Yaskawa INFORM job: kufsatest1_01_01_23_10_57.JBI

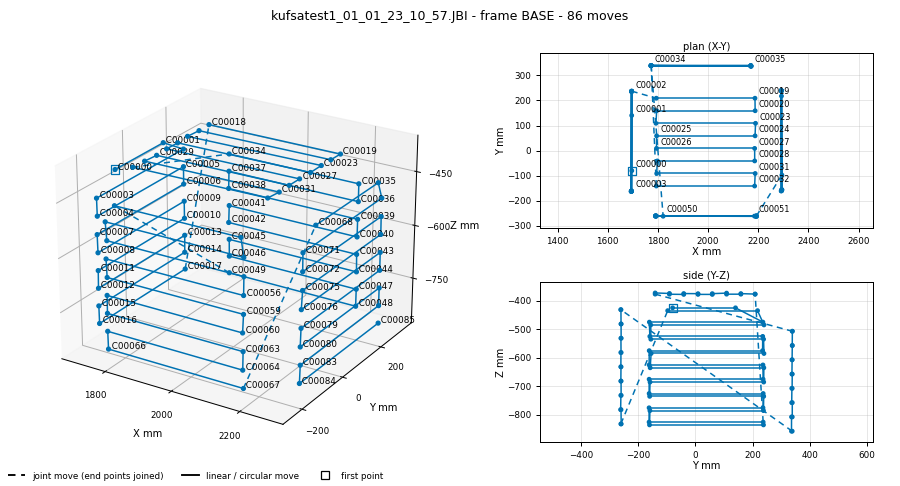
[picture p0: tool path of kufsatest1_01_01_23_10_57.JBI in frame BASE, 86 of 86 moves have a stored position in this frame; points joined in program order, loops and branches not executed]
/JOB
//NAME kufsa_test
//POS
///NPOS 86,0,0,0,0,0
///TOOL 0
///POSTYPE BASE
///RECTAN
///RCONF 1,0,0,0,0,0,0,0,0,0,0,0,0,0,0,0,0,0,0,0,0,0,0,0
C00000=1696.132000,-80.047400,-425.128800,0.000000,90.000000,0.000000
C00001=1695.649900,140.027500,-425.128800,0.000000,90.000000,0.000000
C00002=1695.009700,236.007500,-475.128800,0.000000,90.000000,0.000000
C00003=1694.894300,-161.509200,-475.128800,0.000000,90.000000,0.000000
C00004=1694.500400,-159.876400,-525.128800,0.000000,90.000000,0.000000
C00005=1694.957700,235.269700,-525.128800,0.000000,90.000000,0.000000
C00006=1695.172400,234.870300,-575.128800,0.000000,90.000000,0.000000
C00007=1694.072400,-162.036300,-575.128800,0.000000,90.000000,0.000000
C00008=1695.266200,-162.303200,-625.128800,0.000000,90.000000,0.000000
C00009=1695.465900,236.123700,-625.128800,0.000000,90.000000,0.000000
C00010=1695.422700,236.644700,-675.128800,0.000000,90.000000,0.000000
C00011=1694.457900,-162.352100,-675.128800,0.000000,90.000000,0.000000
C00012=1693.613400,-162.296700,-725.128800,0.000000,90.000000,0.000000
C00013=1695.359600,236.966000,-725.128800,0.000000,90.000000,0.000000
C00014=1695.305600,236.328100,-775.128800,0.000000,90.000000,0.000000
C00015=1693.299800,-162.503900,-775.128800,0.000000,90.000000,0.000000
C00016=1694.079700,-162.510900,-825.128800,0.000000,90.000000,0.000000
C00017=1695.793500,236.889300,-825.128800,0.000000,90.000000,0.000000
C00018=1793.675300,208.803900,-377.180700,-180.000000,0.000000,90.000000
C00019=2187.017900,208.803900,-377.015400,-180.000000,0.000000,90.000000
C00020=2187.698900,158.803900,-375.418500,-180.000000,0.000000,90.000000
C00021=1795.170400,158.803900,-377.409600,-180.000000,0.000000,90.000000
C00022=1792.375400,108.803900,-377.337500,-180.000000,0.000000,90.000000
C00023=2189.165300,108.803900,-373.615200,-180.000000,0.000000,90.000000
C00024=2187.408900,58.803900,-375.476400,-180.000000,0.000000,90.000000
C00025=1795.003900,58.803900,-378.201600,-180.000000,0.000000,90.000000
C00026=1794.543100,8.803900,-378.074400,-180.000000,0.000000,90.000000
C00027=2185.685100,8.803900,-375.544700,-180.000000,0.000000,90.000000
C00028=2185.880000,-41.196100,-375.195400,-180.000000,0.000000,90.000000
C00029=1797.809600,-41.196100,-378.167200,-180.000000,0.000000,90.000000
C00030=1795.305000,-91.196100,-377.541600,-180.000000,0.000000,90.000000
C00031=2187.800700,-91.196100,-374.817700,-180.000000,0.000000,90.000000
C00032=2185.655400,-141.196100,-373.016400,-180.000000,0.000000,90.000000
C00033=1793.794000,-141.196100,-377.211700,-180.000000,0.000000,90.000000
C00034=1773.422800,338.858700,-507.069300,90.000000,0.000000,0.000000
C00035=2170.526400,339.076800,-507.069300,90.000000,0.000000,0.000000
C00036=2170.470000,338.721700,-557.069300,90.000000,0.000000,0.000000
C00037=1772.765600,338.845000,-557.069300,90.000000,0.000000,0.000000
C00038=1772.113800,338.178100,-607.069300,90.000000,0.000000,0.000000
C00039=2169.918900,338.249700,-607.069300,90.000000,0.000000,0.000000
C00040=2169.846800,337.617600,-657.069300,90.000000,0.000000,0.000000
C00041=1773.408600,338.699100,-657.069300,90.000000,0.000000,0.000000
C00042=1771.966000,338.269300,-707.069300,90.000000,0.000000,0.000000
C00043=2169.887200,337.437200,-707.069300,90.000000,0.000000,0.000000
C00044=2170.816100,336.900000,-757.069300,90.000000,0.000000,0.000000
C00045=1773.075800,338.832900,-757.069300,90.000000,0.000000,0.000000
C00046=1773.335100,338.792700,-807.069300,90.000000,0.000000,0.000000
C00047=2171.727500,336.247000,-807.069300,90.000000,0.000000,0.000000
C00048=2171.220400,336.110800,-857.069300,90.000000,0.000000,0.000000
C00049=1773.221800,338.627300,-857.069300,90.000000,0.000000,0.000000
C00050=1820.971900,-261.541800,-431.614400,-90.000000,0.000000,0.000000
C00051=2184.952000,-261.044500,-431.614400,-90.000000,0.000000,0.000000
C00052=2192.839600,-260.681700,-481.614400,-90.000000,0.000000,0.000000
C00053=1791.152000,-260.567100,-481.614400,0.000000,90.000000,0.000000
C00054=1794.425600,-260.324700,-531.614400,-90.000000,0.000000,0.000000
C00055=2193.314000,-261.064500,-531.614400,-90.000000,0.000000,0.000000
C00056=2192.341900,-260.734400,-581.614400,-90.000000,0.000000,0.000000
C00057=1791.071900,-261.005300,-581.614400,-90.000000,0.000000,0.000000
C00058=1793.131800,-261.280300,-631.614400,-90.000000,0.000000,0.000000
C00059=2192.209400,-260.873200,-631.614400,-90.000000,0.000000,0.000000
C00060=2189.954000,-261.359600,-681.614400,-90.000000,0.000000,0.000000
C00061=1791.050300,-260.611400,-681.614400,-90.000000,0.000000,0.000000
C00062=1790.464400,-260.376300,-731.614400,-90.000000,0.000000,0.000000
C00063=2191.354100,-261.246600,-731.614400,-90.000000,0.000000,0.000000
C00064=2190.798500,-262.036100,-781.614400,-90.000000,0.000000,0.000000
C00065=1790.058300,-260.739400,-781.614400,-90.000000,0.000000,0.000000
C00066=1790.686400,-260.189100,-831.614400,-90.000000,0.000000,0.000000
C00067=2192.318900,-261.278300,-831.614400,-90.000000,0.000000,0.000000
C00068=2294.292800,-97.327000,-435.033100,0.000000,0.000000,0.000000
C00069=2292.553200,217.265700,-435.033100,0.000000,0.000000,0.000000
C00070=2291.804400,239.786900,-485.033100,0.000000,0.000000,0.000000
C00071=2294.201800,-156.615000,-485.033100,0.000000,0.000000,0.000000
C00072=2293.933400,-156.359200,-535.033100,0.000000,0.000000,0.000000
C00073=2292.245400,238.334100,-535.033100,0.000000,0.000000,0.000000
C00074=2291.848800,239.682800,-585.033100,0.000000,0.000000,0.000000
C00075=2293.799300,-155.333200,-585.033100,0.000000,0.000000,0.000000
C00076=2292.833100,-158.703500,-635.033100,0.000000,0.000000,0.000000
C00077=2291.947400,239.284200,-635.033100,0.000000,0.000000,0.000000
C00078=2292.084100,238.852100,-685.033100,0.000000,0.000000,0.000000
C00079=2292.973900,-159.159300,-685.033100,0.000000,0.000000,0.000000
C00080=2292.114000,-160.465100,-735.033100,0.000000,0.000000,0.000000
C00081=2291.977800,238.820300,-735.033100,0.000000,0.000000,0.000000
C00082=2292.135300,237.997300,-785.033100,0.000000,0.000000,0.000000
C00083=2292.381400,-159.627800,-785.033100,0.000000,0.000000,0.000000
C00084=2291.307500,-160.899900,-835.033100,0.000000,0.000000,0.000000
C00085=2292.416200,237.973300,-835.033100,0.000000,0.000000,0.000000
//INST
///DATE 2023/01/01 10:55
///ATTR SC,RW,RJ
////FRAME BASE
///GROUP1 RB1
NOP
MOVJ C00000 VJ=15.00
MOVL C00001 V=200.0
MOVL C00002 V=200.0
MOVL C00003 V=200.0
MOVL C00004 V=200.0
MOVL C00005 V=200.0
MOVL C00006 V=200.0
MOVL C00007 V=200.0
MOVL C00008 V=200.0
MOVL C00009 V=200.0
MOVL C00010 V=200.0
MOVL C00011 V=200.0
MOVL C00012 V=200.0
MOVL C00013 V=200.0
MOVL C00014 V=200.0
MOVL C00015 V=200.0
MOVL C00016 V=200.0
MOVL C00017 V=200.0
MOVJ C00018 VJ=15.00
MOVL C00019 V=200.0
MOVL C00020 V=200.0
MOVL C00021 V=200.0
MOVL C00022 V=200.0
MOVL C00023 V=200.0
MOVL C00024 V=200.0
MOVL C00025 V=200.0
MOVL C00026 V=200.0
MOVL C00027 V=200.0
MOVL C00028 V=200.0
MOVL C00029 V=200.0
MOVL C00030 V=200.0
MOVL C00031 V=200.0
MOVL C00032 V=200.0
MOVL C00033 V=200.0
MOVJ C00034 VJ=15.00
MOVL C00035 V=200.0
MOVL C00036 V=200.0
MOVL C00037 V=200.0
MOVL C00038 V=200.0
MOVL C00039 V=200.0
MOVL C00040 V=200.0
MOVL C00041 V=200.0
MOVL C00042 V=200.0
MOVL C00043 V=200.0
MOVL C00044 V=200.0
MOVL C00045 V=200.0
MOVL C00046 V=200.0
MOVL C00047 V=200.0
MOVL C00048 V=200.0
MOVL C00049 V=200.0
MOVJ C00050 VJ=15.00
MOVL C00051 V=200.0
MOVL C00052 V=200.0
MOVL C00053 V=200.0
MOVL C00054 V=200.0
MOVL C00055 V=200.0
MOVL C00056 V=200.0
MOVL C00057 V=200.0
MOVL C00058 V=200.0
MOVL C00059 V=200.0
MOVL C00060 V=200.0
MOVL C00061 V=200.0
MOVL C00062 V=200.0
MOVL C00063 V=200.0
MOVL C00064 V=200.0
MOVL C00065 V=200.0
MOVL C00066 V=200.0
MOVL C00067 V=200.0
MOVJ C00068 VJ=15.00
MOVL C00069 V=200.0
MOVL C00070 V=200.0
MOVL C00071 V=200.0
MOVL C00072 V=200.0
MOVL C00073 V=200.0
MOVL C00074 V=200.0
MOVL C00075 V=200.0
MOVL C00076 V=200.0
MOVL C00077 V=200.0
MOVL C00078 V=200.0
MOVL C00079 V=200.0
MOVL C00080 V=200.0
MOVL C00081 V=200.0
MOVL C00082 V=200.0
MOVL C00083 V=200.0
MOVL C00084 V=200.0
MOVL C00085 V=200.0
END
